TYPE stEntityHeader : STRUCT
    {attribute addProperty Name "Last station"}
    LastStation : enumStations;
    {attribute addProperty Name "Next station"}
    NextStation : enumStations;
END_STRUCT
END_TYPE

(* stored: Version 1.1.0.1, ProductVersion 3.1.4024.6
   DUT stEntityHeader: Id {9bcd5264-dcda-4e6f-a13e-c05fe29274b1} *)
